FUNCTION_BLOCK I_TD (* Time/Date TD *)
  (* Standard: ISO 11783-7; Classification: PGN 65254; Function: Time/Date TD; Description: Copyright (c) 2024 HR Agrartechnik GmbH This program and the accompanying materials are made available under the terms of the Eclipse Public License 2.0 which is available at https://www.eclipse.org/legal/epl-2.0/ SPDX-License-Identifier: EPL-2.0 Message providing current time and date information in the ISOBUS network. https://docs.ms-muc-docs.de/projects/isobus-other-docs/de/latest/PGN/PGN_65254.html *)
  (* Version 1.0, 2024-07-09, Franz Höpfinger, HR Agrartechnik GmbH *)
  PACKAGE isobus::tecu;
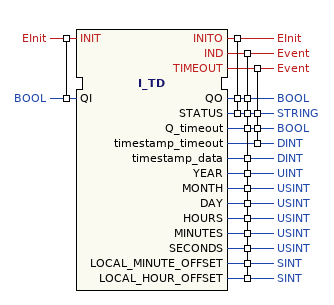
  EVENT_INPUT
    INIT : EInit WITH QI; (* Service Initialization *)
  END_EVENT
  EVENT_OUTPUT
    INITO : EInit WITH QO, STATUS; (* Initialization Confirm *)
    IND WITH QO, timestamp_data, STATUS, Q_timeout, SECONDS, MINUTES, HOURS, MONTH, DAY, YEAR, LOCAL_MINUTE_OFFSET, LOCAL_HOUR_OFFSET; (* Indication from Resource *)
    TIMEOUT WITH timestamp_timeout, STATUS, Q_timeout;
  END_EVENT
  VAR_INPUT
    QI : BOOL; (* Event Input Qualifier *)
  END_VAR
  VAR_OUTPUT
    QO : BOOL; (* Event Output Qualifier *)
    STATUS : STRING;
    Q_timeout : BOOL;
    timestamp_timeout : DINT;
    timestamp_data : DINT;
    YEAR : UINT := UINT#16#FFFF; (* Year (see Attributes for Details) *) {SET_ATTRIBUTE(SPN, 964)} {SET_ATTRIBUTE(SP_Name, 'Year')} {SET_ATTRIBUTE(SP_Position_In_PG, '6')} {SET_ATTRIBUTE(SP_Length, 8)} (* 8 bits *) {SET_ATTRIBUTE(Scaling, '1 y/bit')} {SET_ATTRIBUTE(Offset, 1985)} {SET_ATTRIBUTE(Link, 'https://docs.ms-muc-docs.de/projects/isobus-other-docs/de/latest/PGN/PGN_65254.html#spn-964-year')}
    MONTH : USINT := USINT#16#FF; (* Month (see Attributes for Details) *) {SET_ATTRIBUTE(SPN, 963)} {SET_ATTRIBUTE(SP_Name, 'Month')} {SET_ATTRIBUTE(SP_Position_In_PG, '4')} {SET_ATTRIBUTE(SP_Length, 8)} (* 8 bits *) {SET_ATTRIBUTE(Scaling, '1 month/bit')} {SET_ATTRIBUTE(Offset, 0)} {SET_ATTRIBUTE(Link, 'https://docs.ms-muc-docs.de/projects/isobus-other-docs/de/latest/PGN/PGN_65254.html#spn-963-month')}
    DAY : USINT := USINT#16#FF; (* Day (see Attributes for Details) *) {SET_ATTRIBUTE(SPN, 962)} {SET_ATTRIBUTE(SP_Name, 'Day')} {SET_ATTRIBUTE(SP_Position_In_PG, '5')} {SET_ATTRIBUTE(SP_Length, 8)} (* 8 bits *) {SET_ATTRIBUTE(Scaling, '0.25 d/bit')} {SET_ATTRIBUTE(Offset, 0)} {SET_ATTRIBUTE(Link, 'https://docs.ms-muc-docs.de/projects/isobus-other-docs/de/latest/PGN/PGN_65254.html#spn-962-day')}
    HOURS : USINT := USINT#16#FF; (* Hours (see Attributes for Details) *) {SET_ATTRIBUTE(SPN, 961)} {SET_ATTRIBUTE(SP_Name, 'Hours')} {SET_ATTRIBUTE(SP_Position_In_PG, '3')} {SET_ATTRIBUTE(SP_Length, 8)} (* 8 bits *) {SET_ATTRIBUTE(Scaling, '1 h/bit')} {SET_ATTRIBUTE(Offset, 0)} {SET_ATTRIBUTE(Link, 'https://docs.ms-muc-docs.de/projects/isobus-other-docs/de/latest/PGN/PGN_65254.html#spn-961-hours')}
    MINUTES : USINT := USINT#16#FF; (* Minutes (see Attributes for Details) *) {SET_ATTRIBUTE(SPN, 960)} {SET_ATTRIBUTE(SP_Name, 'Minutes')} {SET_ATTRIBUTE(SP_Position_In_PG, '2')} {SET_ATTRIBUTE(SP_Length, 8)} (* 8 bits *) {SET_ATTRIBUTE(Scaling, '1 min/bit')} {SET_ATTRIBUTE(Offset, 0)} {SET_ATTRIBUTE(Link, 'https://docs.ms-muc-docs.de/projects/isobus-other-docs/de/latest/PGN/PGN_65254.html#spn-960-minutes')}
    SECONDS : USINT := USINT#16#FF; (* Seconds (see Attributes for Details) *) {SET_ATTRIBUTE(SPN, 959)} {SET_ATTRIBUTE(SP_Name, 'Seconds')} {SET_ATTRIBUTE(SP_Position_In_PG, '1')} {SET_ATTRIBUTE(SP_Length, 8)} (* 8 bits *) {SET_ATTRIBUTE(Scaling, '0.25 s/bit')} {SET_ATTRIBUTE(Offset, 0)} {SET_ATTRIBUTE(Link, 'https://docs.ms-muc-docs.de/projects/isobus-other-docs/de/latest/PGN/PGN_65254.html#spn-959-seconds')}
    LOCAL_MINUTE_OFFSET : SINT; (* Local minute offset (see Attributes for Details) *) {SET_ATTRIBUTE(SPN, 1601)} {SET_ATTRIBUTE(SP_Name, 'Local minute offset')} {SET_ATTRIBUTE(SP_Position_In_PG, '7')} {SET_ATTRIBUTE(SP_Length, 8)} (* 8 bits *) {SET_ATTRIBUTE(Scaling, '1 min/bit')} {SET_ATTRIBUTE(Offset, -125)} {SET_ATTRIBUTE(Link, 'https://docs.ms-muc-docs.de/projects/isobus-other-docs/de/latest/PGN/PGN_65254.html#spn-1601-local-minute-offset')}
    LOCAL_HOUR_OFFSET : SINT; (* Local hour offset (see Attributes for Details) *) {SET_ATTRIBUTE(SPN, 1602)} {SET_ATTRIBUTE(SP_Name, 'Local hour offset')} {SET_ATTRIBUTE(SP_Position_In_PG, '8')} {SET_ATTRIBUTE(SP_Length, 8)} (* 8 bits *) {SET_ATTRIBUTE(Scaling, '1 h/bit')} {SET_ATTRIBUTE(Offset, -125)} {SET_ATTRIBUTE(Link, 'https://docs.ms-muc-docs.de/projects/isobus-other-docs/de/latest/PGN/PGN_65254.html#spn-1602-local-hour-offset')}
  END_VAR
END_FUNCTION_BLOCK
